FUNCTION F_DeviceTwin_IsDesiredTopic : BOOL
VAR_INPUT
	sTopic : STRING; // $iothub/twin/PATCH/properties/desired/#	  
END_VAR
VAR
END_VAR

IF FIND(sTopic, '$$iothub/twin/PATCH/properties/desired/') = 0 THEN
	  F_DeviceTwin_IsDesiredTopic := FALSE;
ELSE
	  F_DeviceTwin_IsDesiredTopic := TRUE;
END_IF

END_FUNCTION

(* stored: Version 1.1.0.1, ProductVersion 3.1.4022.3
   POU F_DeviceTwin_IsDesiredTopic: Id {293d9a2c-19a0-4347-b1a4-8e00aa3d0f47}, SpecialFunc None *)
